Fanuc KAREL source: libind_mth.kl

-- Software License Agreement (BSD License)
--
-- Copyright (c) 2012-2014, TU Delft Robotics Institute
-- All rights reserved.
--
-- Redistribution and use in source and binary forms, with or without
-- modification, are permitted provided that the following conditions
-- are met:
--
--  * Redistributions of source code must retain the above copyright
--    notice, this list of conditions and the following disclaimer.
--  * Redistributions in binary form must reproduce the above
--    copyright notice, this list of conditions and the following
--    disclaimer in the documentation and/or other materials provided
--    with the distribution.
--  * Neither the name of the TU Delft Robotics Institute nor the names
--    of its contributors may be used to endorse or promote products
--    derived from this software without specific prior written
--    permission.
--
-- THIS SOFTWARE IS PROVIDED BY THE COPYRIGHT HOLDERS AND CONTRIBUTORS
-- "AS IS" AND ANY EXPRESS OR IMPLIED WARRANTIES, INCLUDING, BUT NOT
-- LIMITED TO, THE IMPLIED WARRANTIES OF MERCHANTABILITY AND FITNESS
-- FOR A PARTICULAR PURPOSE ARE DISCLAIMED. IN NO EVENT SHALL THE
-- COPYRIGHT OWNER OR CONTRIBUTORS BE LIABLE FOR ANY DIRECT, INDIRECT,
-- INCIDENTAL, SPECIAL, EXEMPLARY, OR CONSEQUENTIAL DAMAGES (INCLUDING,
-- BUT NOT LIMITED TO, PROCUREMENT OF SUBSTITUTE GOODS OR SERVICES;
-- LOSS OF USE, DATA, OR PROFITS; OR BUSINESS INTERRUPTION) HOWEVER
-- CAUSED AND ON ANY THEORY OF LIABILITY, WHETHER IN CONTRACT, STRICT
-- LIABILITY, OR TORT (INCLUDING NEGLIGENCE OR OTHERWISE) ARISING IN
-- ANY WAY OUT OF THE USE OF THIS SOFTWARE, EVEN IF ADVISED OF THE
-- POSSIBILITY OF SUCH DAMAGE.


PROGRAM libind_mth
--------------------------------------------------------------------------------
--
-- Shared math functionality
--
-- author: G.A. vd. Hoorn (TU Delft Robotics Institute)
--
--------------------------------------------------------------------------------
%ALPHABETIZE
%COMMENT = 'r2'
%NOBUSYLAMP
%NOLOCKGROUP
%NOPAUSE = COMMAND + TPENABLE + ERROR




--------------------------------------------------------------------------------
--
-- local types & constants
--
--------------------------------------------------------------------------------




--------------------------------------------------------------------------------
--
-- local routine prototypes
--
--------------------------------------------------------------------------------
%INCLUDE include\libind_mth_h




--------------------------------------------------------------------------------
--
-- Empty body
--
--------------------------------------------------------------------------------
BEGIN
END libind_mth




ROUTINE deg_to_rad
BEGIN
	RETURN (r_deg * DEG_2_RAD)
END deg_to_rad




ROUTINE rad_to_deg
BEGIN
	RETURN (r_rad * RAD_2_DEG)
END rad_to_deg




ROUTINE arr_deg2rad
VAR
	len_ : INTEGER
	d_   : INTEGER
BEGIN
	len_ = ARRAY_LEN(a)
	FOR d_ = 1 TO len_ DO
		a[d_] = deg_to_rad(a[d_])
	ENDFOR
END arr_deg2rad




ROUTINE arr_rad2deg
VAR
	len_ : INTEGER
	d_   : INTEGER
BEGIN
	len_ = ARRAY_LEN(a)
	FOR d_ = 1 TO len_ DO
		a[d_] = rad_to_deg(a[d_])
	ENDFOR
END arr_rad2deg


ROUTINE arr2xyzwpr
VAR
	len_ : INTEGER
	d_ : INTEGER
BEGIN
	p.X = a[1] -- mm
	p.Y = a[2] -- mm
	p.Z = a[3] -- mm
	p.W = a[4] -- deg
	p.P = a[5] -- deg
	p.R = a[6] -- deg

	-- reference B-83284JA/02 p.149
	-- Masahiro Furukawa
	p.CONFIG_DATA.CFG_TURN_NO1 = 0
	p.CONFIG_DATA.CFG_TURN_NO2 = 0
	p.CONFIG_DATA.CFG_TURN_NO3 = 0
	p.CONFIG_DATA.CFG_FLIP = FALSE
	p.CONFIG_DATA.CFG_LEFT = FALSE
	p.CONFIG_DATA.CFG_UP = FALSE
	p.CONFIG_DATA.CFG_FRONT = FALSE
END arr2xyzwpr
